Yaskawa INFORM job: AAA.JBI

/JOB
//NAME AAA
//POS
///NPOS 8,0,0,0,0,0
///TOOL 11
///POSTYPE PULSE
///PULSE
C00000=31970,-841,-7031,9752,-64737,-11903
C00001=31970,-841,-7031,9752,-64737,-11903
C00002=31970,-841,-7031,9752,-64737,-11903
C00003=3857,15294,3351,-22976,-60226,-198
C00004=-21617,35142,12009,-51420,-71205,9089
C00005=-21617,35142,12009,-51420,-71205,9089
C00006=-42403,51799,13876,-69358,-88843,13121
C00007=-58721,56844,404,-80660,-106680,14278
//INST
///DATE 2023/04/06 23:24
///ATTR SC,RW
///GROUP1 RB1
NOP
MOVJ C00000 VJ=5.0
TIMER T=1.00
MOVJ C00001 VJ=1.0
TIMER T=0.10
MOVC C00002 V=800.0
MOVC C00003 V=800.0
MOVC C00004 V=800.0 FPT
MOVC C00005 V=800.0
MOVC C00006 V=800.0
MOVC C00007 V=800.0 FPT
END
